PROGRAM MAIN
VAR
	my_variable:REAL;
END_VAR

my_variable:=my_variable-1;

END_PROGRAM

(* stored: Version 1.1.0.1, ProductVersion 3.1.4024.9
   POU MAIN: Id {3306c3db-6852-4c4d-9c38-627bb085fd88}, SpecialFunc None *)
